{attribute 'GeneratedUsingTerminal: EP1816-1008-0016'}
{attribute addProperty BoxType "EP1816-1008-0016"}
{attribute addProperty Id "EtcSlaveTerminalBaseDIG_Inputs_Channel_1AT %I*DIG_Inputs_Channel_38F9DD278DIG_Inputs_Channel_2AT %I*DIG_Inputs_Channel_38F9DD278DIG_Inputs_DeviceAT %I*DIG_Inputs_Device_B3EA42044WcStateAT %I*WcState_9091E0EB2InfoDataAT %I*InfoData_32EB74EA10"}
{attribute addProperty CRC "318247297"}
{attribute addProperty Size "32"}
TYPE EP1816_12F81181 EXTENDS EtcSlaveTerminalBase :
STRUCT
	{attribute addProperty Name "DIG_Inputs_Channel_1"}
	DIG_Inputs_Channel_1 : DIG_Inputs_Channel_38F9DD27;
	{attribute addProperty Name "DIG_Inputs_Channel_2"}
	DIG_Inputs_Channel_2 : DIG_Inputs_Channel_38F9DD27;
	{attribute addProperty Name "DIG_Inputs_Device"}
	DIG_Inputs_Device : DIG_Inputs_Device_B3EA4204;
	{attribute addProperty Name "WcState"}
	WcState : WcState_9091E0EB;
	{attribute addProperty Name "InfoData"}
	InfoData : InfoData_32EB74EA;
END_STRUCT
END_TYPE

(* stored: Version 1.2.0.0, ProductVersion 3.1.4024.9
   DUT EP1816_12F81181: Id {9a212359-1a5a-4e9c-b0fa-97dcee3ad202} *)
